(* IEC 61131-3 sources: Std_PalletMover/Class/AuxHmiWithMqtt, 1 file *)

(* ---- AuxHmiWithMqtt.st ---- *)
(*!
<Class
	Name               = "AuxHmiWithMqtt"
	Revision           = "0.0"
	RealtimeTask       = "false"
	CyclicTask         = "false"
	BackgroundTask     = "false"
	Sigmatek           = "false"
	OSInterface        = "false"
	HighPriority       = "false"
	Automatic          = "false"
	UpdateMode         = "Prescan"
	SharedCommandTable = "true"
	Objectsize         = "(1050,120)">
	<Channels>
		<Server Name="ClassSvr" Visualized="false" Initialize="false" WriteProtected="true" Retentive="false"/>
		<Server Name="HmiInterface" Class="InterfaceAuxHmiMqtt" Visualized="false" Initialize="false" WriteProtected="true" Retentive="false"/>
		<Client Name="ObjCntrlAuxHmi" Required="true" Internal="true"/>
		<Client Name="ObjHimMqttInterface" Required="true" Internal="true"/>
		<Client Name="ObjInterfaceAuxHmiMqtt" Required="true" Internal="true"/>
		<Client Name="op_LogData" Required="false" Internal="false" Comment="Output for logging data to SF_Logger"/>
		<Client Name="p_NextObject" Required="false" Internal="false" Comment="Pointer to next object in linked list"/>
		<Client Name="ToConfiguration" Required="true" Internal="false"/>
		<Client Name="ToSettings" Required="true" Internal="false"/>
		<Client Name="WewoMqtt1" Required="true" Internal="true"/>
		<Client Name="WewoMqtt1_Copy" Required="true" Internal="true"/>
	</Channels>
	<Network Name="AuxHmiWithMqtt">
		<!-- List of Components in this network -->
		<Components>
			<Object
				Name       = "ObjCntrlAuxHmi"
				Class      = "CntrlAuxHmi"
				Position   = "(1260,240)"
				Visualized = "false">
				<Channels>
					<Server Name="AgvState"/>
					<Server Name="ErrorMessage"/>
					<Server Name="ToObject"/>
					<Client Name="op_LogData"/>
					<Client Name="p_NextObject"/>
					<Client Name="ToConfiguration"/>
					<Client Name="ToMqttInterface"/>
					<Client Name="ToSettings"/>
				</Channels>
			</Object>
			<Object
				Name       = "ObjHimMqttInterface"
				Class      = "MqttInterface"
				Position   = "(1260,720)"
				Visualized = "true"
				Remotely   = "true">
				<Channels>
					<Server Name="ClassSvr"/>
					<Server Name="ErrorCnt"/>
					<Server Name="InterfaceState"/>
					<Server Name="LastErrorCode"/>
					<Client Name="op_LogData"/>
				</Channels>
			</Object>
			<Object
				Name       = "ObjInterfaceAuxHmiMqtt"
				Class      = "InterfaceAuxHmiMqtt"
				Position   = "(4230,690)"
				Visualized = "false">
				<Channels>
					<Server Name="ClassSvr"/>
				</Channels>
			</Object>
			<Object
				Name       = "WewoMqtt1"
				Class      = "WewoMqtt"
				Position   = "(2670,270)"
				Visualized = "true"
				Remotely   = "true">
				<Channels>
					<Server Name="DataString"/>
					<Server Name="GrantedQoS"/>
					<Server Name="PublishInterval" Value="10 sec"/>
					<Server Name="QoS"/>
					<Server Name="RetainData"/>
					<Server Name="TopicItem" Value="&quot;ErrorMessage&quot;"/>
					<Server Name="TopicName"/>
					<Server Name="TopicPath" Value="&quot;Hmi&quot;"/>
					<Server Name="TopicState"/>
					<Server Name="TopicType" Value="MQTTTopic::MT_Publish_OnChange"/>
					<Client Name="ocMQTTClient_Interface"/>
					<Client Name="op_LogData"/>
				</Channels>
			</Object>
			<Object
				Name       = "WewoMqtt1_Copy"
				Class      = "WewoMqtt"
				Position   = "(2670,990)"
				Visualized = "true"
				Remotely   = "true">
				<Channels>
					<Server Name="DataString"/>
					<Server Name="GrantedQoS"/>
					<Server Name="PublishInterval" Value="10 sec"/>
					<Server Name="QoS"/>
					<Server Name="RetainData"/>
					<Server Name="TopicItem" Value="&quot;ErrorMessage&quot;"/>
					<Server Name="TopicName"/>
					<Server Name="TopicPath" Value="&quot;Hmi&quot;"/>
					<Server Name="TopicState"/>
					<Server Name="TopicType" Value="MQTTTopic::MT_Publish_OnChange"/>
					<Client Name="ocMQTTClient_Interface"/>
					<Client Name="op_LogData"/>
				</Channels>
			</Object>
		</Components>
		<Comments>
		</Comments>
		<!-- List of Connections in this network -->
		<Connections>
			<Connection Source="this.ObjCntrlAuxHmi" Destination="ObjCntrlAuxHmi.ToObject"/>
			<Connection Source="this.ObjHimMqttInterface" Destination="ObjHimMqttInterface.ClassSvr"/>
			<Connection Source="this.WewoMqtt1" Destination="WewoMqtt1.TopicState"/>
			<Connection Source="WewoMqtt1.ocMQTTClient_Interface" Destination="ObjHimMqttInterface.InterfaceState" Vertices="(2670,360),(2236,870),"/>
			<Connection Source="ObjCntrlAuxHmi.ToMqttInterface" Destination="ObjHimMqttInterface.ClassSvr" Vertices="(1260,570),(2236,810),"/>
			<Connection Source="ObjCntrlAuxHmi.ToSettings" Destination="this.ToSettings" Vertices="(1260,510),(38,330),"/>
			<Connection Source="ObjCntrlAuxHmi.ToConfiguration" Destination="this.ToConfiguration" Vertices="(1260,450),(38,270),"/>
			<Connection Source="ObjHimMqttInterface.op_LogData" Destination="this.op_LogData" Vertices="(1260,810),(38,390),"/>
			<Connection Source="this.ObjInterfaceAuxHmiMqtt" Destination="ObjInterfaceAuxHmiMqtt.ClassSvr"/>
			<Connection Source="ObjCntrlAuxHmi.p_NextObject" Destination="this.p_NextObject" Vertices="(1260,390),(38,210),"/>
			<Connection Source="this.WewoMqtt1_Copy" Destination="WewoMqtt1_Copy.TopicState"/>
			<Connection Source="WewoMqtt1_Copy.ocMQTTClient_Interface" Destination="ObjHimMqttInterface.InterfaceState" Vertices="(2670,1080),(2236,870),"/>
			<Connection Source="this.HmiInterface" Destination="ObjInterfaceAuxHmiMqtt.ClassSvr" Vertices="(5228,270),(5056,780),"/>
		</Connections>
		<!-- Headerfiles -->
		<Options>
		</Options>
	</Network>
</Class>
*)
AuxHmiWithMqtt : CLASS
  //Servers:
	ClassSvr 	: SvrChCmd_DINT;
	HmiInterface 	: SvrChCmd_DINT;
  //Clients:
	ObjCntrlAuxHmi 	: CltChCmd_CntrlAuxHmi;
	ObjHimMqttInterface 	: CltChCmd_MqttInterface;
	WewoMqtt1 	: CltChCmd_WewoMqtt;
	p_NextObject 	: CltChCmd_LinkedObjectBase;
	ToConfiguration 	: CltChCmd_AgvConfig;
	ToSettings 	: CltChCmd_AgvSettings;
	op_LogData 	: CltCh_gpt_LogData;
	WewoMqtt1_Copy 	: CltChCmd_WewoMqtt;
	ObjInterfaceAuxHmiMqtt 	: CltChCmd_InterfaceAuxHmiMqtt;
  //Variables:
  //Functions:

	FUNCTION VIRTUAL GLOBAL HmiInterface::Read
		VAR_OUTPUT
			output (EAX) 	: DINT;
		END_VAR;
  //Tables:
	FUNCTION @STD
		VAR_OUTPUT
			ret_code	: CONFSTATES;
		END_VAR;
	FUNCTION GLOBAL TAB @CT_;
END_CLASS;

#pragma using CntrlAuxHmi
#pragma using InterfaceAuxHmiMqtt
#pragma using MqttInterface
#pragma using WewoMqtt
#pragma usingLtd AgvConfig
#pragma usingLtd AgvSettings
#pragma usingLtd LinkedObjectBase

FUNCTION VIRTUAL GLOBAL AuxHmiWithMqtt::HmiInterface::Read
	VAR_OUTPUT
		output (EAX) 	: DINT;
	END_VAR

	HmiInterface := ObjInterfaceAuxHmiMqtt.ClassSvr.Read();
	output := HmiInterface;

END_FUNCTION
